PROGRAM MAIN
VAR
	HeaterRatio			:REAL	:= 20;
	FanRatio			:REAL;
	Region				:REAL	:= 2.5; //Allowed error +- for the steady-state
	
	fbTempScale			:fbScale;
	fbFControl			:fbFuzzyController;
	fbPIControl			:fbPIContoller;
	
	Timer				:TON;
END_VAR

//Handle digital I/O
SLL(SteadyStateRegion := Region);

//HeaterRatio can be cnaged from the GUI
IO.AO1_Heater := REAL_TO_INT(27468 * HeaterRatio/100);
//Used in the GUI
FanRatio := INT_TO_REAL(IO.AO0_Fan)/INT_TO_REAL(27468)*100;


//Run the controller
//Controller can be switched between PI and Fuzzy
IF SLL.ControllerSwitch THEN
	//Longer samplingtime allows error to accumulate
	//10ms had too small changes between samples
	Timer(IN := NOT Timer.Q, PT := T#0.1S);
	IF Timer.Q THEN
		fbFControl(On := SLL.ControllerOn);
	END_IF
ELSE
	fbPIControl(On := SLL.ControllerOn);
END_IF

//Current temperature as celsius
fbTempScale(IN := IO.AI0_Temp, Scale_L := 20, Scale_H := 120);
Temperatures.T_Act := fbTempScale.OUT;

END_PROGRAM

(* stored: Version 1.1.0.1, ProductVersion 3.1.4022.6
   POU MAIN: Id {178d1884-1f61-4494-864d-b432efcec7a1}, SpecialFunc None *)
